{region '#Template'}
	{attribute 'Version' := '5.0.0.0'}
	{attribute 'Tags' := '"LCID": "1031", "Text": "Automatisierungssteuerung, Gerät, Einstellungen, Systemzeit, BACnet Adapter Zeit"'}
	{attribute 'Tags' := '"LCID": "1033", "Text": "Automation control, Device, Settings, Systemzeit, BACnet Adapter Time"'}
	{attribute 'Using' := '"Type": "Template", "URI": "SysTime"'}		 		 
	{attribute 'Description' := '"LCID": "1031", "Text": "BACnet Adapter Zeit abrufen und lokal setzen"'}
	{attribute 'Description' := '"LCID": "1033", "Text": "Get BACnet Adapter Time and set locally"'}
{endregion}

FUNCTION_BLOCK FB_BA_BACnetTime_TO_SysTime
VAR_INPUT
END_VAR
VAR_OUTPUT
END_VAR
VAR_INPUT CONSTANT PERSISTENT	
	sExternalAmsNetId						: T_AmsNetId := ''; // Beispiel,Example: '192.168.131.1.1.1'
	{attribute 'parameterUnit':= 's'}
	GetBACnetAdapterTime_nTiAuto			: UDINT := 600;
	{attribute 'parameterUnit':= 's'}
	GetLocalSysTime_nTiAuto					: UDINT := 60;
END_VAR	
VAR_INPUT CONSTANT
	GetExtSysTime				: FB_BA_GetTime;

	SetSysTimeLocal				: FB_BA_SetTime;
	SetBACnetAdapterTime		: FB_BA_SetBACnetAdapterTime;

	GetLocalSysTime				: FB_BA_GetTime;
	GetBACnetAdapterTime		: FB_BA_GetBACnetAdapterTime;
END_VAR
VAR
	GetExtSysTime_bSync					: BOOL;	
	GetExtSysTime_rtrigSync				: R_TRIG;
	
	GetBACnetAdapterTime_wYear				: WORD;
	GetBACnetAdapterTime_wMonth				: WORD;
	GetBACnetAdapterTime_wDayOfWeek			: WORD;
	GetBACnetAdapterTime_wDay				: WORD;
	GetBACnetAdapterTime_wHour				: WORD;
	GetBACnetAdapterTime_wMinute			: WORD;
	GetBACnetAdapterTime_wSecond			: WORD;
	GetBACnetAdapterTime_wMilliseconds		: WORD;		
	
	// F_BA_STDateTime_TO_TIMESTRUCT
END_VAR

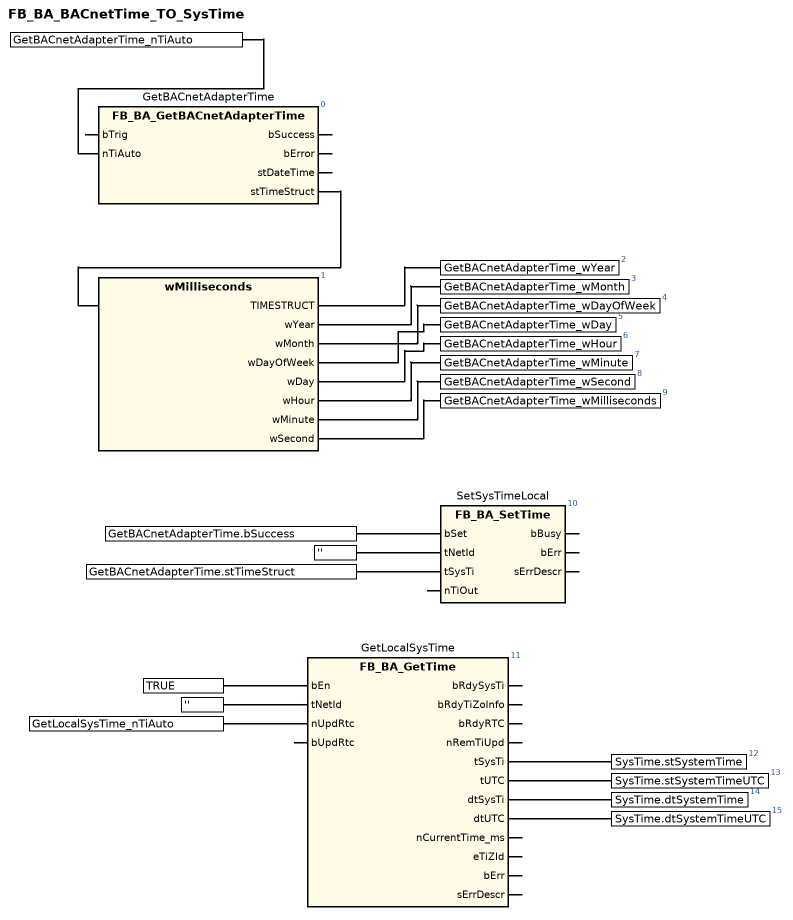
GetBACnetAdapterTime(nTiAuto := GetBACnetAdapterTime_nTiAuto); // FB_BA_GetBACnetAdapterTime
GetBACnetAdapterTime_wYear := GetBACnetAdapterTime.stTimeStruct.TIMESTRUCT;
GetBACnetAdapterTime_wMonth := GetBACnetAdapterTime.stTimeStruct.wYear;
GetBACnetAdapterTime_wDayOfWeek := GetBACnetAdapterTime.stTimeStruct.wMonth;
GetBACnetAdapterTime_wDay := GetBACnetAdapterTime.stTimeStruct.wDayOfWeek;
GetBACnetAdapterTime_wHour := GetBACnetAdapterTime.stTimeStruct.wDay;
GetBACnetAdapterTime_wMinute := GetBACnetAdapterTime.stTimeStruct.wHour;
GetBACnetAdapterTime_wSecond := GetBACnetAdapterTime.stTimeStruct.wMinute;
GetBACnetAdapterTime_wMilliseconds := GetBACnetAdapterTime.stTimeStruct.wSecond;
SetSysTimeLocal(
    bSet := GetBACnetAdapterTime.bSuccess,
    tNetId := '',
    tSysTi := GetBACnetAdapterTime.stTimeStruct); // FB_BA_SetTime
GetLocalSysTime(bEn := TRUE, tNetId := '', nUpdRtc := GetLocalSysTime_nTiAuto); // FB_BA_GetTime
SysTime.stSystemTime := GetLocalSysTime.tSysTi;
SysTime.stSystemTimeUTC := GetLocalSysTime.tUTC;
SysTime.dtSystemTime := GetLocalSysTime.dtSysTi;
SysTime.dtSystemTimeUTC := GetLocalSysTime.dtUTC;

END_FUNCTION_BLOCK

(* stored: Version 1.1.0.1, ProductVersion 3.1.4024.12
   POU FB_BA_BACnetTime_TO_SysTime: Id {a16a60a9-9bfc-4672-8d4f-8747a543a78d}, SpecialFunc None *)
